Fanuc KAREL source: IO0057.KL

-- PROVISIONAL review KL for V940-1; original PC SHA256 a0b359f87ee51ef9ac07ab06030a469c1f9aca34c730a23a64dd81ae55763215
-- Incomplete behavior may be omitted. Consult companion uncertainty JSON. Do not deploy.
PROGRAM IO0057
%NOLOCKGROUP
-- UNRESOLVED_LOCAL_POOL 5 cells at code offset 13; source declarations unknown
-- DIRECT_LOCAL_WORD_ACCESS alone does not prove INTEGER, REAL, or BOOLEAN
BEGIN
  -- V9_ZERO_TABLE_METADATA_HINT layout=0001; no indexed target words; source/name/runtime held
  -- V9_ZERO_GLOBAL_LAYOUT_HINT count-one $GROUP table, zero relocation slots, two routine descriptors; executable preamble and source held
  -- V9_SIGNAL_ARRAY_LITERAL_HINT GOUT direct_index_literal_write index_cell=40
  -- UNRESOLVED_PC offsets 0-18; opcodes 2B,2C,7B
  -- UNRESOLVED_PC offsets 23-30; opcodes 9D,23
  -- UNRESOLVED_PC offsets 35-49; opcodes 2E,22,9D,33,35
  -- UNRESOLVED_PC offsets 54-61; opcodes 9D,23
  -- UNRESOLVED_PC offsets 66-77; opcodes 2E,23
  -- UNRESOLVED_PC offsets 82-91; opcodes 9D,21,1A
  -- UNRESOLVED_PC offsets 96-100; opcodes 7F
  -- UNRESOLVED_PC offsets 105-109; opcodes 27,AA
  -- UNRESOLVED_PC offsets 114-118; opcodes 7F
END IO0057
